FUNCTION_BLOCK HMIUpdate
VAR_INPUT
	
END_VAR
VAR_OUTPUT
END_VAR
VAR
	i : INT;
	LoopCounter : INT;
	UltimateByPassCounter : INT;
	
	
	
	Active: INT;
END_VAR



GVL_HMI.GlobalFault_Code := MAIN.GlobalEstopCode;

IF MAIN.GlobalEstopActive THEN
	LoopCounter := LoopCounter + 1;
	ELSE
	loopcounter := 0;
END_IF

IF LoopCounter = 0 OR LoopCounter > 400 THEN
	GVL_HMI.EstopLight := TRUE;
END_IF

IF LoopCounter > 800 THEN
	LoopCounter := 0;
	GVL_HMI.EstopLight := FALSE;
END_IF

GVL_HMI.Patient1.AgeTimer(IN:= NOT GVL_HMI.Patient1.ActiveSwitch, PT:= T#5S, ET=>GVL_HMI.Patient1.AGE);
GVL_HMI.Patient2.AgeTimer(IN:= NOT GVL_HMI.Patient2.ActiveSwitch, PT:= T#5S, ET=>GVL_HMI.Patient2.AGE);
GVL_HMI.Patient3.AgeTimer(IN:= NOT GVL_HMI.Patient3.ActiveSwitch, PT:= T#5S, ET=>GVL_HMI.Patient3.AGE);
GVL_HMI.Patient4.AgeTimer(IN:= NOT GVL_HMI.Patient4.ActiveSwitch, PT:= T#5S, ET=>GVL_HMI.Patient4.AGE);
 GVL_HMI.Patient1.ActiveSwitch := FALSE;
 GVL_HMI.Patient2.ActiveSwitch:= FALSE;
//IF NOT GVL_HMI.Patient2.ActiveSwitch THEN GVL_HMI.Patient2.ActiveSwitch := TRUE; END_IF
//IF NOT GVL_HMI.Patient3.ActiveSwitch THEN GVL_HMI.Patient3.ActiveSwitch:= TRUE; END_IF
GVL_HMI.Patient3.ActiveSwitch:= FALSE;
GVL_HMI.Patient4.ActiveSwitch:= FALSE;
//IF NOT GVL_HMI.Patient4.ActiveSwitch THEN GVL_HMI.Patient4.ActiveSwitch:= TRUE; END_IF


GVL_HMI.JoyStick1ScreenStateCommanded := main.SerialRemoteNear.ScreenCommanded;
GVL_HMI.JoyStick2ScreenStateCOmmanded := MAIN.SerialRemoteFar.ScreenCommanded;
GVL_HMI.JoyStick1DeadManState := main.SerialRemoteNear.DeadmanPressed>0;
GVL_HMI.JoyStick2DeadManState := MAIN.SerialRemoteFar.DeadmanPressed>0;
GVL_HMI.Joystick1ZAxisPressed := MAIN.SerialRemoteNear.ZAxisPressed>0;
GVL_HMI.JoyStick2ZAxisPressed :=MAIN.SerialRemoteFar.ZAxisPressed>0;
GVL_HMI.JoyStick1SyncPressed := MAIN.SerialRemoteNear.SyncPressed>0;
GVL_HMI.JoyStick2SyncPressed:= MAIN.SerialRemoteFar.SyncPressed>0;
GVL_HMI.JoyStick1Estop := main.SerialRemoteNear.EstopPressed>0;
GVL_HMI.Joystick2Estop := MAIN.SerialRemoteFar.EstopPressed>0;
GVL_HMI.JoyStick1Age := MAIN.SerialRemoteNear.Age;
GVL_HMI.JoyStick2Age := MAIN.SerialRemoteFar.Age;

END_FUNCTION_BLOCK

(* stored: Version 1.1.0.1, ProductVersion 3.1.4022.3
   POU HMIUpdate: Id {e90bd3c8-d3fe-4341-b760-c678d5af554e}, SpecialFunc None *)
